FUNCTION Convert_DT_TO_TOD : Hresult
VAR_INPUT
	in : DT;
	out : REFERENCE TO TOD;
END_VAR
VAR
	converted : TOD;
END_VAR

converted := DT_TO_TOD(in);

IF (TOD_TO_DT(converted) <> in) THEN
	Convert_DT_TO_TOD := INCOMPATIBLE;
	RETURN;
END_IF

out := converted;

END_FUNCTION

(* stored: Version 1.1.0.1, ProductVersion 3.1.4024.12
   POU Convert_DT_TO_TOD: Id {8a680c2f-5121-4f1d-86ac-9563e029f969}, SpecialFunc None *)
